INTERFACE I_REFERENCE_TO EXTENDS I_Datatype

PROPERTY PUBLIC IsValidReference : BOOL
GET
END_GET
END_PROPERTY

END_INTERFACE

(* stored: Version 1.1.0.1, ProductVersion 3.1.4026.18
   Itf I_REFERENCE_TO: Id {d58f73ff-1d4c-05a4-2ba1-ac397ce5e773}
   Property IsValidReference: Id {0531ddf0-0b9c-0b03-05ee-bf10c0d34c5b}
   Get Get: Id {a6776383-d9a7-0b6b-2d9a-056dc735e256} *)
